// TwinCAT 3 PLC project PRG_B_ActuatorDecorator
// Title: B_ActuatorDecorator
// Company: RafalOS
// Author: Rafał Osajda
// ProjectVersion: 0.0.0.3
// ProgramVersion: 3.1.4024.0
// libraries:
//   B_Actuator, * (RafalOS)
//   B_Base, * (RafalOS)
//   B_BaseDecorate, * (RafalOS)
//   B_IO, * (RafalOS)
//   B_IODecorator, * (RafalOS)
//   Tc2_Standard, * (Beckhoff Automation GmbH)
//   Tc2_System, * (Beckhoff Automation GmbH)
//   Tc3_Module, * (Beckhoff Automation GmbH)
// project tree:
//   / PlcTask.TcTTO
//   POUs Compilation/ PRG_Compilation.TcPOU
//   POUs/ FB_ActuatorDecoratorTest.TcPOU, FB_ActuatorDecoratorTestWithoutTime.TcPOU, FB_ActuatorDecoratorTestWithTime.TcPOU, ITF_ActuatorDecoratorTest.TcIO (not stored)

CONFIGURATION PRG_B_ActuatorDecorator
    RESOURCE PLC ON TwinCAT3
        TASK PlcTask(INTERVAL := T#10ms, PRIORITY := 20);
        PROGRAM PRG_Compilation WITH PlcTask : PRG_Compilation;
    END_RESOURCE
END_CONFIGURATION

// ---- POUs Compilation/PRG_Compilation.TcPOU
PROGRAM PRG_Compilation
VAR
	senActuator1Start			: FB_Sensor_NO;
	senActuator1End				: FB_Sensor_NO;
	evActuator1Control			: FB_Electrovalve_5on3_2Coil_Vented;
	fbActuator1					: FB_Actuator (
									senStart		:= senActuator1Start,
									senEnd			:= senActuator1End,
									evControl		:= evActuator1Control
								);
								
	senActuator1StartDecoratorTest	: FB_SensorNODecoratorTest (fbToDecorate := senActuator1Start);
	senActuator1EndDecoratorTest	: FB_SensorNODecoratorTest (fbToDecorate := senActuator1End);
	
	fbActuator1DecoratorTest	: FB_ActuatorDecoratorTest (
									fbToDecorate 	:= fbActuator1,
									actActuator		:= fbActuator1,
									senStart		:= senActuator1StartDecoratorTest,
									senEnd		:= senActuator1EndDecoratorTest
								);

	fbActuator1DecoratorTestWithoutTime	: FB_ActuatorDecoratorTestWithoutTime (
									fbToDecorate 	:= fbActuator1,
									actActuator		:= fbActuator1,
									senStart		:= senActuator1StartDecoratorTest,
									senEnd		:= senActuator1EndDecoratorTest
								);

	fbActuator1DecoratorTestWithTime	: FB_ActuatorDecoratorTestWithTime (
									fbToDecorate 	:= fbActuator1,
									actActuator		:= fbActuator1,
									senStart		:= senActuator1StartDecoratorTest,
									senEnd		:= senActuator1EndDecoratorTest
								);
	
END_VAR

END_PROGRAM

// ---- POUs/FB_ActuatorDecoratorTest.TcPOU
FUNCTION_BLOCK FB_ActuatorDecoratorTest EXTENDS FB_BaseControlElementDecoratorParent IMPLEMENTS ITF_ActuatorDecoratorTest
VAR
	itfactActuator		: ITF_Actuator;
	itfsenStart			: ITF_SensorDecoratorTest;
	itfsenEnd			: ITF_SensorDecoratorTest;

	itfczStart			: ITF_SensorDecoratorTest;		//przypisanie czujnika z pozycji startowej w czasie przesuwania w testach
	itfczStop			: ITF_SensorDecoratorTest;		//przypisanie czujnika z pozycji końcowej w czasie przesuwania w testach

	iStepTestCycle		: INT := 0;

	
END_VAR

METHOD FB_init : BOOL
VAR_INPUT
	bInitRetains : BOOL; // if TRUE, the retain variables are initialized (warm start / cold start)
	bInCopyCode : BOOL;  // if TRUE, the instance afterwards gets moved into the copy code (online change)
	fbToDecorate		: ITF_DecoratedElement;
	actActuator			: ITF_Actuator;
	senStart			: ITF_SensorDecoratorTest;
	senEnd				: ITF_SensorDecoratorTest;
	
END_VAR
THIS^.itfactActuator	:= actActuator;
THIS^.itfsenStart		:= senStart;
THIS^.itfsenEnd			:= senEnd;
END_METHOD

METHOD IsEnd : BOOL
VAR_INPUT
END_VAR
IsEnd		:= THIS^.itfactActuator.IsEnd ();
END_METHOD

METHOD PUBLIC IsStart : BOOL
VAR_INPUT
END_VAR
IsStart		:= THIS^.itfactActuator.IsStart ();
END_METHOD

(*			
	EVERDE sp. z o.o.
	Rafał Osajda		31.03.2025		TC 4024.66
	Uruchomienie cyklu przesuwania do początku
*)
METHOD PUBLIC MoveToEnd
VAR_INPUT
END_VAR
THIS^.itfactActuator.MoveToEnd ();
END_METHOD

(*			
	EVERDE sp. z o.o.
	Rafał Osajda		31.03.2025		TC 4024.66
	Uruchomienie cyklu przesuwania do początku
*)
METHOD PUBLIC MoveToStart
VAR_INPUT
END_VAR
THIS^.itfactActuator.MoveToStart ();
END_METHOD

METHOD PUBLIC MovingToEndBusy : BOOL
VAR_INPUT
END_VAR
MovingToEndBusy		:= THIS^.itfactActuator.MovingToEndBusy ();
END_METHOD

METHOD PUBLIC MovingToEndFirstCycyle : BOOL
VAR_INPUT
END_VAR
MovingToEndFirstCycyle		:= THIS^.itfactActuator.MovingToEndFirstCycyle ();
END_METHOD

METHOD PUBLIC MovingToEndStatus : BOOL
VAR_INPUT
END_VAR
MovingToEndStatus		:= THIS^.itfactActuator.MovingToEndStatus ();
END_METHOD

METHOD PUBLIC MovingToStartBusy : BOOL
VAR_INPUT
END_VAR
MovingToStartBusy		:= THIS^.itfactActuator.MovingToStartBusy ();
END_METHOD

METHOD PUBLIC MovingToStartFirstCycle : BOOL
VAR_INPUT
END_VAR
MovingToStartFirstCycle 	:= THIS^.itfactActuator.MovingToStartFirstCycle ();
END_METHOD

METHOD PUBLIC MovingToStartStatus : BOOL
VAR_INPUT
END_VAR
MovingToStartStatus		:= THIS^.itfactActuator.MovingToStartStatus ();
END_METHOD

END_FUNCTION_BLOCK

// ---- POUs/FB_ActuatorDecoratorTestWithoutTime.TcPOU
FUNCTION_BLOCK FB_ActuatorDecoratorTestWithoutTime EXTENDS FB_ActuatorDecoratorTest
VAR

END_VAR

(*			
	EVERDE sp. z o.o.
	Rafał Osajda		27.03.2025		TC 4024.66
	Wywolanie co cykl operacji 
*)
METHOD PUBLIC ExecuteEveryCycle_Operation
VAR_INPUT
END_VAR
//testować czy jest cykl przesuwania do gdzieś i po czasie uruchamiać lub wyłączać czujniki 
THIS^.itfactActuator.ExecuteEveryCycle_Operation ();

IF (THIS^.itfactActuator.MovingToStartFirstCycle ()) THEN
	THIS^.itfczStart		:= THIS^.itfsenEnd;
	THIS^.itfczStop			:= THIS^.itfsenStart;
	THIS^.iStepTestCycle	:= 10;
END_IF

IF (THIS^.itfactActuator.MovingToEndFirstCycyle ()) THEN
	THIS^.itfczStart		:= THIS^.itfsenStart;
	THIS^.itfczStop			:= THIS^.itfsenEnd;
	THIS^.iStepTestCycle	:= 10;
END_IF

CASE THIS^.iStepTestCycle OF
10	: THIS^.iStepTestCycle	:= THIS^.iStepTestCycle + 10;	//pierwszy cykl
20	: THIS^.iStepTestCycle	:= THIS^.iStepTestCycle + 10;
30	: 
	THIS^.itfczStart.SetContract (bIN := FALSE); 
	THIS^.iStepTestCycle	:= THIS^.iStepTestCycle + 10;
40	: 
	THIS^.itfczStop.SetContract (bIN := TRUE);
	THIS^.iStepTestCycle	:= 0;
END_CASE
END_METHOD

END_FUNCTION_BLOCK

// ---- POUs/FB_ActuatorDecoratorTestWithTime.TcPOU
FUNCTION_BLOCK FB_ActuatorDecoratorTestWithTime EXTENDS FB_ActuatorDecoratorTest
VAR
	tonSensorTurnOffTime	: Tc2_Standard.TON;
	tonSensorTurnOnTime		: Tc2_Standard.TON;

END_VAR

(*			
	EVERDE sp. z o.o.
	Rafał Osajda		27.03.2025		TC 4024.66
	Wywolanie co cykl operacji 
*)
METHOD PUBLIC ExecuteEveryCycle_Operation
VAR_INPUT
END_VAR
//testować czy jest cykl przesuwania do gdzieś i po czasie uruchamiać lub wyłączać czujniki 
THIS^.itfactActuator.ExecuteEveryCycle_Operation();
THIS^.tonSensorTurnOffTime ();
THIS^.tonSensorTurnOnTime ();

IF (THIS^.itfactActuator.MovingToStartFirstCycle ()) THEN
	THIS^.itfczStart			:= THIS^.itfsenEnd;
	THIS^.itfczStop				:= THIS^.itfsenStart;
	THIS^.tonSensorTurnOffTime.PT	:= REAL_TO_TIME (THIS^.itfactActuator.ParameterGetValue (1) * 0.1);
	THIS^.tonSensorTurnOffTime.IN	:= TRUE;
	THIS^.tonSensorTurnOnTime.PT	:= REAL_TO_TIME (THIS^.itfactActuator.ParameterGetValue (1) * 0.7);
	THIS^.iStepTestCycle		:= 10;
END_IF

IF (THIS^.itfactActuator.MovingToEndFirstCycyle ()) THEN
	THIS^.itfczStart			:= THIS^.itfsenStart;
	THIS^.itfczStop				:= THIS^.itfsenEnd;
	THIS^.tonSensorTurnOffTime.PT	:= REAL_TO_TIME (THIS^.itfactActuator.ParameterGetValue (2) * 0.1);
	THIS^.tonSensorTurnOffTime.IN	:= TRUE;
	THIS^.tonSensorTurnOnTime.PT	:= REAL_TO_TIME (THIS^.itfactActuator.ParameterGetValue (2) * 0.7);
	THIS^.iStepTestCycle		:= 10;
END_IF

CASE THIS^.iStepTestCycle OF
10	: IF (THIS^.tonSensorTurnOffTime.Q) THEN
		THIS^.tonSensorTurnOffTime.IN	:= FALSE;
		THIS^.itfczStart.SetContract (bIN := FALSE);
		THIS^.tonSensorTurnOnTime.IN	:= TRUE;
		iStepTestCycle		:= THIS^.iStepTestCycle + 10;
	END_IF
20	: IF (THIS^.tonSensorTurnOnTime.Q) THEN
		THIS^.tonSensorTurnOnTime.IN	:= FALSE;
		THIS^.itfczStop.SetContract (bIN := TRUE);
		THIS^.iStepTestCycle	:= 0;
	END_IF
END_CASE
END_METHOD

END_FUNCTION_BLOCK
